PROGRAM FBDsRULE
VAR
	nothingspecial : BOOL;
	
END_VAR

// NETWORK 1

END_PROGRAM

(* stored: Version 1.1.0.1, ProductVersion 3.1.4024.12
   POU FBDsRULE: Id {463221a7-1b25-47bd-a4e2-e6b491046b2a}, SpecialFunc None *)
